FUNCTION_BLOCK FB_ILK_TEST
VAR_INPUT
END_VAR
VAR_OUTPUT
END_VAR
VAR
END_VAR

END_FUNCTION_BLOCK

(* stored: Version 1.1.0.1, ProductVersion 3.1.4022.18
   POU FB_ILK_TEST: Id {e6f9e748-aea7-4235-8fb2-3876556b20bc}, SpecialFunc None *)
